{attribute 'qualified_only'}
VAR_GLOBAL CONSTANT
	eInternalLog			: E_LogLevel := E_LogLevel.eInfo;	(* min. log level for internal logging. *)
	nBufferLen 				: UINT := 8192;		(* Length of per task log buffer in bytes *)
	nMaxScopedContext		: UINT := 4;		(* Max. number of nested scope context. *)
	eMaxLogLevel			: E_LogLevel := E_LogLevel.eWarn;
END_VAR

(* stored: Version 1.1.0.1, ProductVersion 3.1.4024.13
   GVL Config: Id {a1726ba6-7c08-42a0-82ef-a943824dc09f}, ParameterList True *)
